FUNCTION_BLOCK LargeSortingConveyor EXTENDS Conveyor
VAR_INPUT
END_VAR
VAR_OUTPUT
END_VAR
VAR
	m_rampPusherStart : MonostableCylinder;
	m_rampPusherMid : MonostableCylinder;
	m_Switch : Switch;
	
	m_presenceSensorStart : PresenceSensor;
	m_opticalSensorStart : OpticalSensor;
	m_opticalSensorMid : OpticalSensor;
	m_opticalSensorEnd : OpticalSensor;
	m_inductiveSensorStart : InductiveSensor;
	m_inductiveSensorMid : InductiveSensor;
	
	m_rampStart : Ramp;
	m_rampMiddle : Ramp;
	m_rampEnd : Ramp;
END_VAR

PROPERTY LightWPAtEnd : BOOL
GET
LightWPAtEnd := m_opticalSensorEnd.Value;
END_GET
END_PROPERTY

PROPERTY LightWPAtMid : BOOL
GET
LightWPAtMid := m_opticalSensorMid.Value;
END_GET
END_PROPERTY

PROPERTY LightWPAtStart : BOOL
GET
LightWPAtStart := m_opticalSensorStart.Value;
END_GET
END_PROPERTY

PROPERTY MetalWPAtMid : BOOL
GET
MetalWPAtMid := m_inductiveSensorMid.Value;
END_GET
END_PROPERTY

PROPERTY MetalWPAtStart : BOOL
GET
MetalWPAtStart := m_inductiveSensorStart.Value;
END_GET
END_PROPERTY

METHOD METH_Ramp1Pusher_Extend : BOOL
VAR_INPUT
END_VAR
m_rampPusherStart.METH_Extend();
END_METHOD

METHOD METH_Ramp1Pusher_Retract : BOOL
VAR_INPUT
END_VAR
m_rampPusherStart.METH_Retract();
END_METHOD

METHOD METH_Ramp2Pusher_Extend : BOOL
VAR_INPUT
END_VAR
m_rampPusherMid.METH_Extend();
END_METHOD

METHOD METH_Ramp2Pusher_Retract : BOOL
VAR_INPUT
END_VAR
m_rampPusherMid.METH_Retract();
END_METHOD

METHOD METH_Switch_Extend : BOOL
VAR_INPUT
END_VAR
m_Switch.METH_Extend();
END_METHOD

METHOD METH_Switch_Retract : BOOL
VAR_INPUT
END_VAR
m_Switch.METH_Retract();
END_METHOD

PROPERTY WPAtRampEnd : BOOL
GET
WPAtRampEnd := m_rampEnd.m_presenceSensorRampFull.Value;
END_GET
END_PROPERTY

PROPERTY WPAtRampMiddle : BOOL
GET
WPAtRampMiddle := m_rampMiddle.m_presenceSensorRampFull.Value;
END_GET
END_PROPERTY

PROPERTY WPAtRampStart : BOOL
GET
WPAtRampStart := m_rampStart.m_presenceSensorRampFull.Value;
END_GET
END_PROPERTY

PROPERTY WPAtStart : BOOL
GET
WPAtStart := m_presenceSensorStart.Value;
END_GET
END_PROPERTY

END_FUNCTION_BLOCK

(* stored: Version 1.1.0.1
   POU LargeSortingConveyor: Id {a79cbb88-76ef-4a13-a238-fa308bd8c032}, SpecialFunc None
   Folder Methods: Id {c6437f9a-27b7-4cc0-a8d4-cb7b10ef5b3c}
   Folder Properties: Id {9b639b1e-89df-422a-8b35-4f64cf0abf1b}
   Property LightWPAtEnd: Id {70f5ef49-760f-40f0-8a6a-910b31bf3038}
   Get Get: Id {3db4633f-5262-43ea-bb5b-5e6c3fb25343}
   Property LightWPAtMid: Id {3e6ef8e7-a914-4230-b17c-d08117d0cfaa}
   Get Get: Id {a6849aed-f8bb-4430-9ac7-e9a78e14b8f0}
   Property LightWPAtStart: Id {dcd8ed8b-3a3e-4349-8cdc-b96ccd55c9d7}
   Get Get: Id {ca47d8d3-7577-4f7d-b049-415c23dbf254}
   Property MetalWPAtMid: Id {dfd0aa66-617a-4b7a-a88d-30dc1793c45c}
   Get Get: Id {6f5760b6-bff4-4c59-9feb-f7732fac2554}
   Property MetalWPAtStart: Id {aed07a49-5e83-422c-929d-9088beb392a0}
   Get Get: Id {68f56475-d6af-4fd7-bd0b-569ad3bc47bb}
   Method METH_Ramp1Pusher_Extend: Id {c89c6de8-c6d0-4098-962a-07724390c605}
   Method METH_Ramp1Pusher_Retract: Id {540eb60e-9a37-429a-bd99-9dc85a1b0f91}
   Method METH_Ramp2Pusher_Extend: Id {1961b9b6-9846-40fe-8fb7-365d75560222}
   Method METH_Ramp2Pusher_Retract: Id {c85925f4-a910-46ac-8fb7-600566fc9aeb}
   Method METH_Switch_Extend: Id {32f4abfc-ef2c-45a1-85e3-c1989c168180}
   Method METH_Switch_Retract: Id {0b902dec-a348-4ae3-b4ec-6d7be7271fbe}
   Property WPAtRampEnd: Id {edb6102d-633f-4f3e-97fb-baf0b2661b3c}
   Get Get: Id {eec8ab5c-bef9-4687-8617-6c6c11e147fe}
   Property WPAtRampMiddle: Id {14d2008d-3425-4363-961a-0eed315949df}
   Get Get: Id {40b88a62-d605-47c2-ba01-cb2d750fac7a}
   Property WPAtRampStart: Id {e2d93316-a242-43ae-a8b0-1f9170ee72a7}
   Get Get: Id {37107552-44a3-43ae-8be5-16419118e5c9}
   Property WPAtStart: Id {9079270e-93fa-4573-b2db-64bf784f3e74}
   Get Get: Id {f27dcc24-002e-4d57-b264-5845e6e31d31} *)
